FUNCTION FB_CountConv : REAL
VAR_INPUT
	COUNTS_IN 			: DINT;
END_VAR
VAR
END_VAR
VAR_OUTPUT
	MEASC_OUT 			: REAL;
	MEASF_OUT 			: REAL;
END_VAR

// Conversion for counts to mm -> distance [resolution (nm) * (nm -> mm) * # of counts]

// Renishaw DIP-SWITCH CONFIG, 12/09/20
// NOTE: CONSULT RENISHAW USER MANUAL FOR SWITCH SETTING CONFIGURATION BREAKDOWN

// Switch Up   Switch Down
//    [0]		  [-]
//    [-]         [o]
//
// 15               1
// [ooo-o---|o--o-o--]
// [---o-ooo|-oo-o-oo]

// Coarse resolution conversion
MEASC_OUT := 79 * 0.000001 * COUNTS_IN;

// Fine resolution conversion
MEASF_OUT := 39.5 * 0.000001 * COUNTS_IN;

END_FUNCTION

(* stored: Version 1.1.0.1, ProductVersion 3.1.4024.2
   POU FB_CountConv: Id {1e807885-6745-4d98-882c-3aa7e1b57558}, SpecialFunc None *)
